Universal Robots PolyScope program: Dovetail_buttom.urp

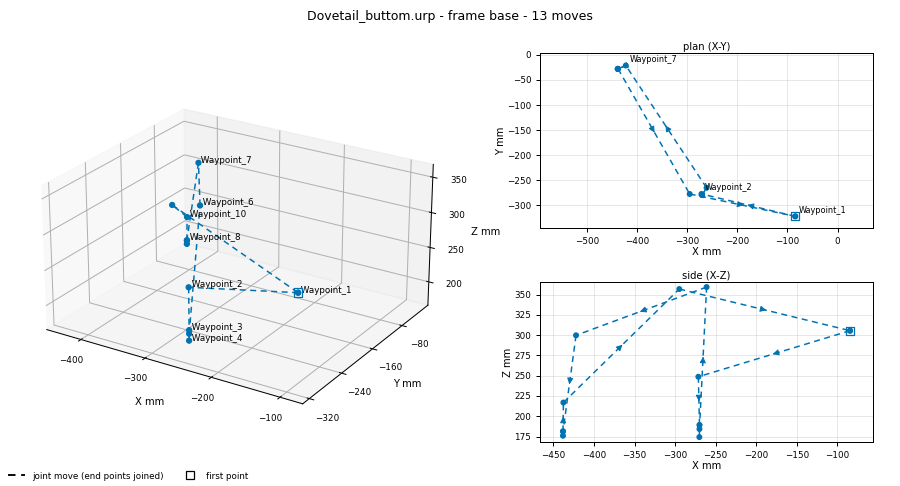
[picture p0: tool path of Dovetail_buttom.urp in frame base, 13 of 13 moves have a stored position in this frame; points joined in program order, loops and branches not executed]
Program Dovetail_buttom (installation=default directory=/programs/usbdisk/Zahra1 createdIn=5.11.11.1010533 lastSavedIn=5.11.11.1010533 robotSerialNumber=20205300864)
Calibrated DH parameters: a=[-0.000166, -0.243494, -0.153108, 0.000057, -0.000123, 0]; d=[0.151897, -1.34267, 53.988124, -52.514559, 0.085283, 0.092193]; alpha=[1.572472, -0.003756, 0.002824, 1.570807, -1.572621, 0]; deltaTheta=[0, 0.020704, 7.033215, -0.770746, 0.000004, 0]
Robot Program (runOnlyOnce=true)
  MoveJ speed 60 deg/s, acceleration 80 deg/s^2 (useActiveTCP=true) feature=Base
    Waypoint Waypoint_1: TCP in base x=-84.299 y=-321.875 z=305.481 mm, rx=-2.0809 ry=-2.2572 rz=0.0984 rad; joints [-79.978, -91.201, -87.971, -91.7, 84.671, 815.506] deg
    URCap Gripper (Robotiq_Grippers, Robotiq Inc.) dataModel(position=40.3921568627451, force=97.0, speed=52.0, positionInDouble=40.3921568627451, forceInDouble=97.0, speedInDouble=52.0, slaveIds=[9], blocking=true, robotCompliant=false)
    Waypoint Waypoint_2: TCP in base x=-271.331 y=-277.245 z=248.685 mm, rx=2.1395 ry=2.2708 rz=0.0333 rad; joints [-115.145, -107.434, -84.034, -79.202, 91.534, 781.557] deg
    Waypoint Waypoint_3: TCP in base x=-269.925 y=-279.225 z=189.342 mm, rx=-2.2148 ry=-2.2212 rz=0.0183 rad; joints [-114.324, -111.587, -95.684, -62.097, 89.49, 785.661] deg
    Waypoint Waypoint_4: TCP in base x=-270.095 y=-279.3 z=174.311 mm, rx=-2.2149 ry=-2.2212 rz=0.0183 rad; joints [-114.35, -113.356, -97.651, -58.356, 89.492, 785.648] deg
    URCap Gripper (Robotiq_Grippers, Robotiq Inc.) dataModel(position=76.58823529411765, force=97.0, speed=52.0, positionInDouble=76.58823529411765, forceInDouble=97.0, speedInDouble=52.0, slaveIds=[9], blocking=true, robotCompliant=false)
    Waypoint Waypoint_5: TCP in base x=-269.973 y=-279.25 z=184.246 mm, rx=-2.2149 ry=-2.2212 rz=0.0183 rad; joints [-114.333, -112.162, -96.381, -60.822, 89.495, 785.659] deg
    Waypoint Waypoint_6: TCP in base x=-261.14 y=-264.906 z=359.27 mm, rx=2.2115 ry=2.193 rz=-0.0528 rad; joints [-114.22, -102.925, -61.164, -103.443, 90.669, 786.347] deg
    Waypoint Waypoint_7: TCP in base x=-422.159 y=-21.173 z=299.802 mm, rx=-2.1803 ry=-2.2414 rz=0.0412 rad; joints [-159.112, -114.533, -61.195, -92.45, 89.809, 739.377] deg
    Waypoint Waypoint_8: TCP in base x=-438.191 y=-27.917 z=181.366 mm, rx=-2.2293 ry=-2.2118 rz=0.0272 rad; joints [-159.18, -123.839, -78.786, -66.335, 90.279, 741.395] deg
    Waypoint Waypoint_9: TCP in base x=-438.261 y=-27.999 z=175.934 mm, rx=-2.2292 ry=-2.2119 rz=0.0271 rad; joints [-159.175, -124.37, -79.469, -65.126, 90.28, 741.399] deg
    URCap Gripper (Robotiq_Grippers, Robotiq Inc.) dataModel(position=38.431372549019606, force=97.0, speed=52.0, positionInDouble=38.431372549019606, forceInDouble=97.0, speedInDouble=52.0, slaveIds=[9], blocking=true, robotCompliant=false)
    Waypoint Waypoint_8: TCP in base x=-438.191 y=-27.917 z=181.366 mm, rx=-2.2293 ry=-2.2118 rz=0.0272 rad; joints [-159.18, -123.839, -78.786, -66.335, 90.279, 741.395] deg
    Waypoint Waypoint_10: TCP in base x=-437.737 y=-27.494 z=216.888 mm, rx=-2.2293 ry=-2.2117 rz=0.0272 rad; joints [-159.199, -120.99, -73.409, -74.561, 90.278, 741.364] deg
    Waypoint Waypoint_11: TCP in base x=-294.805 y=-277.288 z=356.828 mm, rx=-1.8865 ry=-2.467 rz=-0.0298 rad; joints [-117.454, -114.271, -44.517, -112.545, 88.059, 767.431] deg
    Waypoint Waypoint_1: TCP in base x=-84.299 y=-321.875 z=305.481 mm, rx=-2.0809 ry=-2.2572 rz=0.0984 rad; joints [-79.978, -91.201, -87.971, -91.7, 84.671, 815.506] deg
